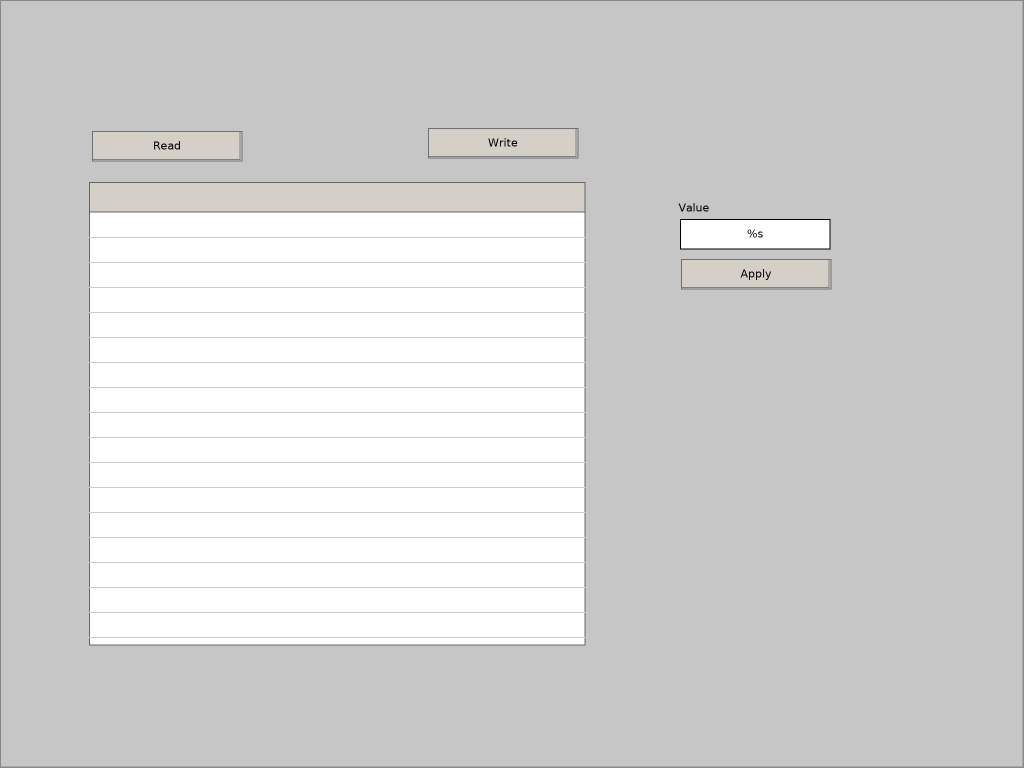
VISUALIZATION MaS_800_SettingScreen  // 1024x768
    Frame (0,0 1024x768)
        shows Tmp_000_Template(header := gHMIData.hmiHeader)
    Table (89,182 496x463), data array: MachineSettings.Setting
        p1420305297: MachineSettings.varSelectedColumn
        p4052804203: MachineSettings.varSelectedColumnValid
        p1137915858: MachineSettings.varSelectedRow
        p1822360349: MachineSettings.varSelectedRowValid
        p1128707560: MachineSettings.numElementsOfSettings
        p3854506369: MachineSettings.Setting[INDEX].TextName
        p1892666644: MachineSettings.Setting[INDEX].Value
        p338671338: MachineSettings.Setting[INDEX].hasChanged
        Columns.Column.[1].Template: OnMouseClick: execute { MachineSettings.numSelectedSettingNew := MachineSettings.Setting[MachineSettings.varSelectedRow].Value }
    Button (92,131 150x30), "Read"
        tap MachineSettings.btnRead
    Button (428,128 150x30), "Write"
        tap MachineSettings.btnWrite
    Label (619,193 150x30), "Value"
    Rectangle (680,219 150x30), "%s", text variable: MachineSettings.numSelectedSettingNew
        OnMouseClick: OpenDialog Dialog=dialogEnterValueInteger, Parameters={enteredValue: MachineSettings.numSelectedSettingNew}, Selected={1: }, OpenModal=True, OpenCentered=True
    Button (681,259 150x30), "Apply"
        tap MachineSettings.btnMoveValue
END_VISUALIZATION

(* stored: Version 1.1.0.1, ProductVersion 3.1.4024.11
   Visu MaS_800_SettingScreen: Id {44f1c459-314b-01ad-1879-0976785968a8} *)
